PROGRAM MAIN
VAR
END_VAR

GVL_IO.dOut_1:=GVL_IO.ACK;

END_PROGRAM

(* stored: Version 1.1.0.1, ProductVersion 3.1.4022.17
   POU MAIN: Id {200bc85e-1c1e-4948-a108-a3c502c86435}, SpecialFunc None *)
